FUNCTION_BLOCK JADEDestroyerFB (* JADE Destroyer *)
  (* Standard: 61499-1 *)
  (* Version 1.0, 2010-04-22, AnLo, TUT *)
  (* Compiler header: package fb.rt; *)
  (* Compiler Java Sun JDK 1.5.0 *)
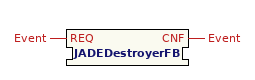
  EVENT_INPUT
    REQ; (* Normal Execution Request *)
  END_EVENT
  EVENT_OUTPUT
    CNF; (* Execution Confirmation *)
  END_EVENT
END_FUNCTION_BLOCK
